// TIA Portal V18 export
FUNCTION "MotionController" : Void   // FC14, LAD
{ S7_Optimized_Access := 'TRUE' }
AUTHOR : HenriP
VERSION : 0.1
// stored: AutoNumber true, IsIECCheckEnabled false, SetENOAutomatically false, UDAEnableTagReadback false
   VAR_INPUT
      "E-STOP" : Bool;
      JogPBtn : Bool;
      JogNBtn : Bool;
      TargetRange : DInt;
      PosMax : DInt;
      PosMin : DInt;
      AxisColision : Bool;
      DoorSensor : Bool;
   END_VAR
   VAR_OUTPUT
      AxisOutput : Struct
         DriveEnabled : Bool;
         Ready : Bool;
         Warning : Bool;
         Fault : Bool;
         SupplyVoltPresent : Bool;
         ControlFCT_HMI : Bool;
         StateOPM : Int;
         HaltNotActive : Bool;
         AckStart : Bool;
         MC : Bool;
         AckTeach : Bool;
         DriveMoving : Bool;
         DragError : Bool;
         StandStillControl : Bool;
         HomingValid : Bool;
         ActualRecordNo : Int;
         RC1 : Bool;
         RCC : Bool;
         VelocityLimitReached : Bool;
         StrokeLimitReached : Bool;
         FunctionIsActive : Bool;
         ActualFunctionNumber : Int;
         ActualFunctionGroup : Int;
         ActualPosition : DInt;
         ActualVelocity : DInt;
         ActualForce : DInt;
         ActualRotRamp : DInt;
         ActualRotSpeed : DInt;
      END_STRUCT;
      TargetReached : Bool;
      Overange : Bool;
   END_VAR
   VAR_IN_OUT
      AxisInput : Struct
         EnableDrive : Bool;
         Stop : Bool;
         Halt : Bool;
         Brake : Bool;
         ResetFault : Bool;
         HMIAccessLocked : Bool;
         OPM : Int;
         StartTask : Bool;
         StartHoming : Bool;
         JogPos : Bool;
         JogNeg : Bool;
         TeachActValue : Bool;
         ClearRemPos : Bool;
         Relative : Bool;
         DeactivateStrokeLimit : Bool;
         ExecuteFunction : Bool;
         RecordNo : Int;
         SetFunctionNumber : Int;
         SetFunctionGroup : Int;
         SetValueVelocity : DInt;
         SetValuePosition : DInt;
         SetValueForceRamp : DInt;
         SetValueForce : DInt;
         SetValueRotRamp : DInt;
         SetValueRotSpeed : DInt;
      END_STRUCT;
      FestoDB : "FHPP_CTRL";
      TaskE : Bool;
      TaskM : Bool;
   END_VAR
   VAR_TEMP
      TargetDistance : DInt;
      ErrorValue : Int;
      Pos : DInt;
      PosAdd : DInt;
      PosSub : DInt;
      TaskEBis : Bool;
      JogPOv : DInt;
   END_VAR
   VAR_TEMP   // added for the SCL form of the ladder/FBD networks
      _w1 : Bool;
      _w2 : Bool;
   END_VAR
BEGIN

REGION Network 1: Enable Axis - Stop Control
   // For safety reason the Safety torque control is on a special loop , Emergency stop may move there too
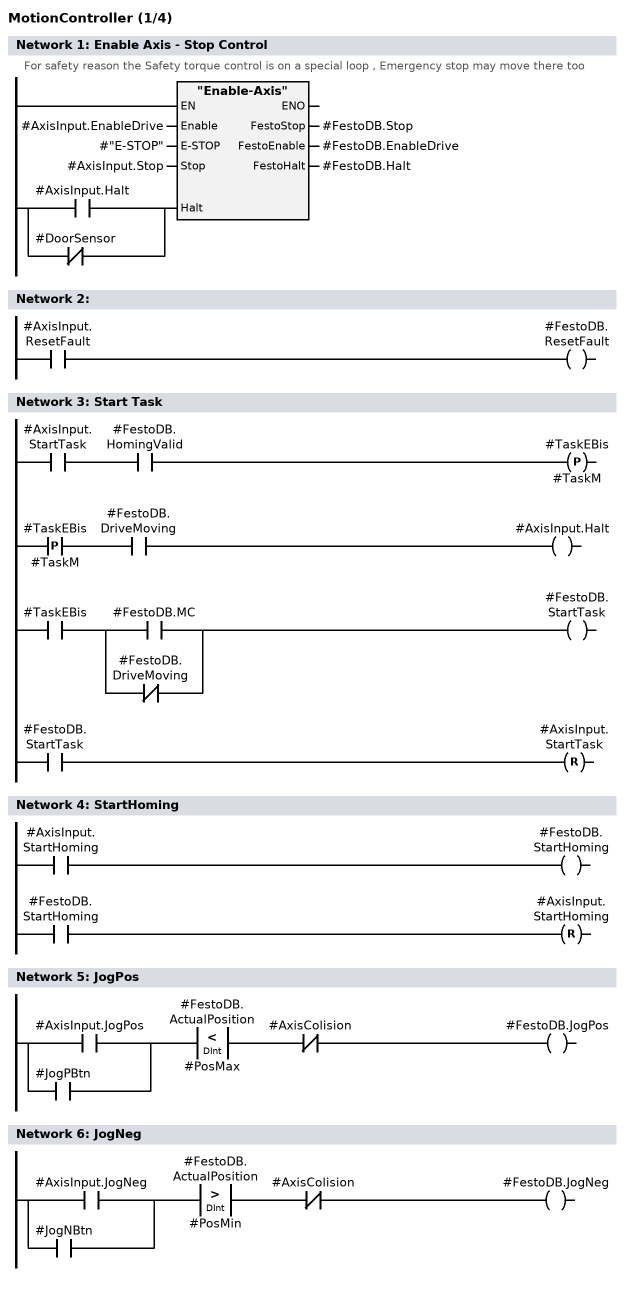
   RUNG wire#powerrail
      "Enable-Axis"(Halt := wire#w1, Enable := #AxisInput.EnableDrive, "E-STOP" := #"E-STOP", Stop := #AxisInput.Stop, FestoStop => #FestoDB.Stop, FestoEnable => #FestoDB.EnableDrive, FestoHalt => #FestoDB.Halt)
   END_RUNG
   RUNG wire#powerrail
      Contact( #AxisInput.Halt )
   END_RUNG wire#w1
   RUNG wire#powerrail
      I_Contact( #DoorSensor )
   END_RUNG wire#w1
   // the same network as SCL:
   "Enable-Axis"(Enable := #AxisInput.EnableDrive,
                 "E-STOP" := #"E-STOP",
                 Stop := #AxisInput.Stop,
                 Halt := #AxisInput.Halt OR NOT #DoorSensor,
                 FestoStop => #FestoDB.Stop,
                 FestoEnable => #FestoDB.EnableDrive,
                 FestoHalt => #FestoDB.Halt);
END_REGION

REGION Network 2
   RUNG wire#powerrail
      Contact( #AxisInput.ResetFault )
      Coil( #FestoDB.ResetFault )
   END_RUNG
   // the same network as SCL:
   #FestoDB.ResetFault := #AxisInput.ResetFault;
END_REGION

REGION Network 3: Start Task
   #_w1 := #AxisInput.StartTask AND #FestoDB.HomingValid;
   #TaskEBis := #_w1 AND NOT #TaskM;   // rising edge
   #TaskM := #_w1;
   #_w2 := #TaskEBis AND NOT #TaskM;   // rising edge of #TaskEBis
   #TaskM := #TaskEBis;
   #AxisInput.Halt := #_w2 AND #FestoDB.DriveMoving;
   #FestoDB.StartTask := #TaskEBis AND (#FestoDB.MC OR NOT #FestoDB.DriveMoving);
   IF #FestoDB.StartTask THEN #AxisInput.StartTask := FALSE; END_IF;
END_REGION

REGION Network 4: StartHoming
   RUNG wire#powerrail
      Contact( #AxisInput.StartHoming )
      Coil( #FestoDB.StartHoming )
   END_RUNG
   RUNG wire#powerrail
      Contact( #FestoDB.StartHoming )
      R_Coil( #AxisInput.StartHoming )
   END_RUNG
   // the same network as SCL:
   #FestoDB.StartHoming := #AxisInput.StartHoming;
   IF #FestoDB.StartHoming THEN #AxisInput.StartHoming := FALSE; END_IF;
END_REGION

REGION Network 5: JogPos
   RUNG wire#powerrail
      Contact( #AxisInput.JogPos )
      wire#w1
      { S7_Templates := "SrcType := DInt" } LT_Contact(in1 := #FestoDB.ActualPosition, in2 := #PosMax)
      I_Contact( #AxisColision )
      Coil( #FestoDB.JogPos )
   END_RUNG
   RUNG wire#powerrail
      Contact( #JogPBtn )
   END_RUNG wire#w1
   // the same network as SCL:
   #FestoDB.JogPos := (#AxisInput.JogPos OR #JogPBtn) AND (#FestoDB.ActualPosition < #PosMax) AND NOT #AxisColision;
END_REGION

REGION Network 6: JogNeg
   RUNG wire#powerrail
      Contact( #AxisInput.JogNeg )
      wire#w1
      { S7_Templates := "SrcType := DInt" } GT_Contact(in1 := #FestoDB.ActualPosition, in2 := #PosMin)
      I_Contact( #AxisColision )
      Coil( #FestoDB.JogNeg )
   END_RUNG
   RUNG wire#powerrail
      Contact( #JogNBtn )
   END_RUNG wire#w1
   // the same network as SCL:
   #FestoDB.JogNeg := (#AxisInput.JogNeg OR #JogNBtn) AND (#FestoDB.ActualPosition > #PosMin) AND NOT #AxisColision;
END_REGION

REGION Network 7: Relative Input Command
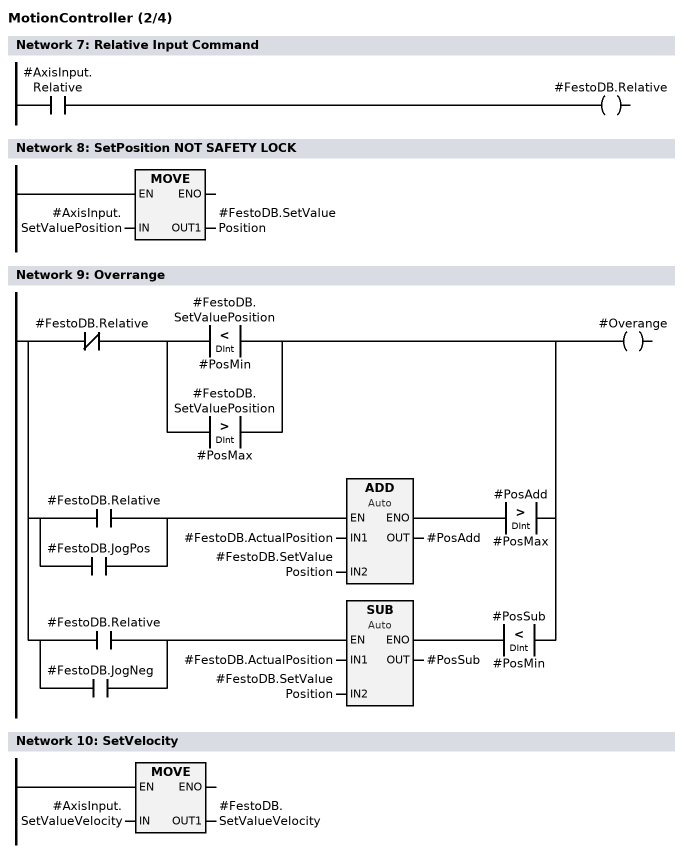
   RUNG wire#powerrail
      Contact( #AxisInput.Relative )
      Coil( #FestoDB.Relative )
   END_RUNG
   // the same network as SCL:
   #FestoDB.Relative := #AxisInput.Relative;
END_REGION

REGION Network 8: SetPosition NOT SAFETY LOCK
   RUNG wire#powerrail
      Move(in := #AxisInput.SetValuePosition, out1 => #FestoDB.SetValuePosition)
   END_RUNG
   // the same network as SCL:
   #FestoDB.SetValuePosition := #AxisInput.SetValuePosition;
END_REGION

REGION Network 9: Overrange
   RUNG wire#powerrail
      I_Contact( #FestoDB.Relative )
      wire#w1
      { S7_Templates := "SrcType := DInt" } LT_Contact(in1 := #FestoDB.SetValuePosition, in2 := #PosMin)
      wire#w2
      Coil( #Overange )
   END_RUNG
   RUNG wire#w1
      { S7_Templates := "SrcType := DInt" } GT_Contact(in1 := #FestoDB.SetValuePosition, in2 := #PosMax)
   END_RUNG wire#w2
   RUNG wire#powerrail
      Contact( #FestoDB.Relative )
      wire#w3
      Add(in1 := #FestoDB.ActualPosition, in2 := #FestoDB.SetValuePosition, out => #PosAdd)
      { S7_Templates := "SrcType := DInt" } GT_Contact(in1 := #PosAdd, in2 := #PosMax)
   END_RUNG wire#w2
   RUNG wire#powerrail
      Contact( #FestoDB.JogPos )
   END_RUNG wire#w3
   RUNG wire#powerrail
      Contact( #FestoDB.Relative )
      wire#w4
      Sub(in1 := #FestoDB.ActualPosition, in2 := #FestoDB.SetValuePosition, out => #PosSub)
      { S7_Templates := "SrcType := DInt" } LT_Contact(in1 := #PosSub, in2 := #PosMin)
   END_RUNG wire#w2
   RUNG wire#powerrail
      Contact( #FestoDB.JogNeg )
   END_RUNG wire#w4
   // the same network as SCL:
   #_w1 := #FestoDB.Relative OR #FestoDB.JogPos;
   IF #_w1 THEN #PosAdd := #FestoDB.ActualPosition + #FestoDB.SetValuePosition; END_IF;
   #_w2 := #FestoDB.Relative OR #FestoDB.JogNeg;
   IF #_w2 THEN #PosSub := #FestoDB.ActualPosition - #FestoDB.SetValuePosition; END_IF;
   #Overange := (NOT #FestoDB.Relative AND ((#FestoDB.SetValuePosition < #PosMin) OR (#FestoDB.SetValuePosition > #PosMax))) OR (#_w1 AND (#PosAdd > #PosMax)) OR (#_w2 AND (#PosSub < #PosMin));
END_REGION

REGION Network 10: SetVelocity
   RUNG wire#powerrail
      Move(in := #AxisInput.SetValueVelocity, out1 => #FestoDB.SetValueVelocity)
   END_RUNG
   // the same network as SCL:
   #FestoDB.SetValueVelocity := #AxisInput.SetValueVelocity;
END_REGION

REGION Network 11: Output Feedback
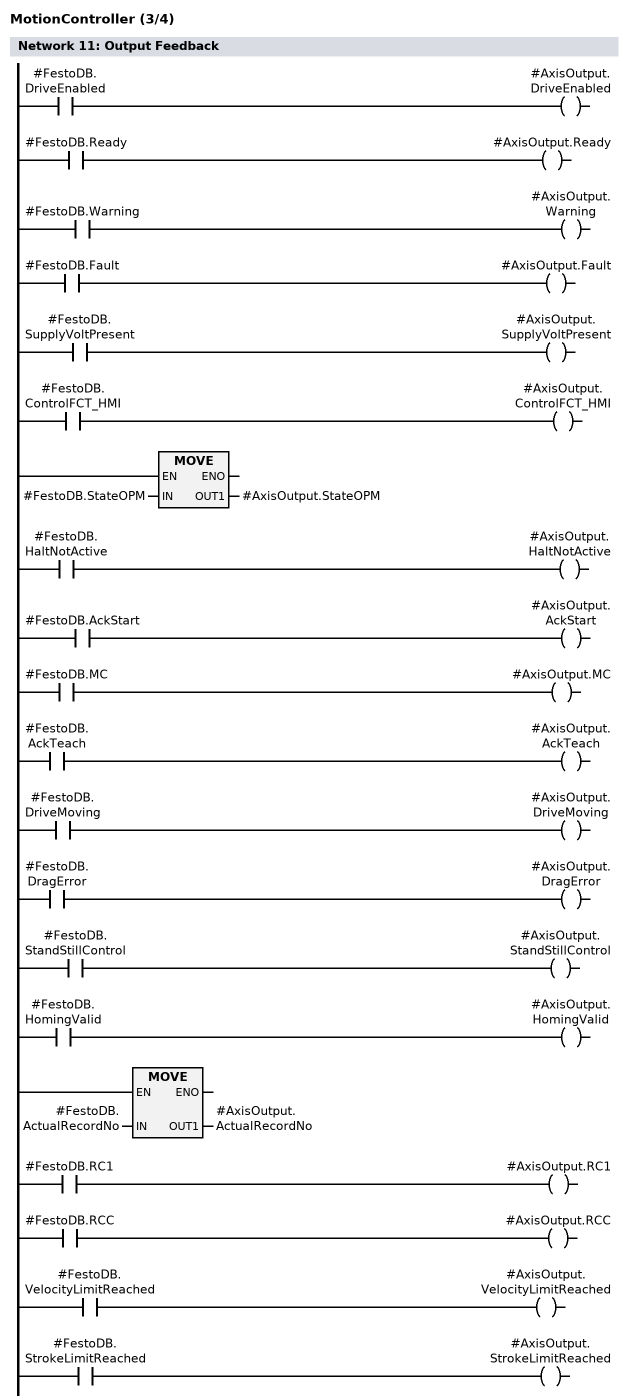
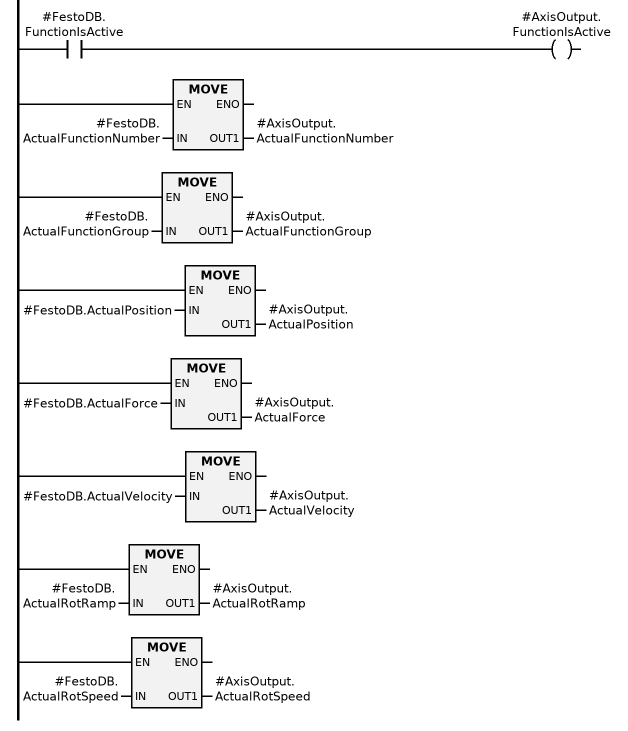
   RUNG wire#powerrail
      Contact( #FestoDB.DriveEnabled )
      Coil( #AxisOutput.DriveEnabled )
   END_RUNG
   RUNG wire#powerrail
      Contact( #FestoDB.Ready )
      Coil( #AxisOutput.Ready )
   END_RUNG
   RUNG wire#powerrail
      Contact( #FestoDB.Warning )
      Coil( #AxisOutput.Warning )
   END_RUNG
   RUNG wire#powerrail
      Contact( #FestoDB.Fault )
      Coil( #AxisOutput.Fault )
   END_RUNG
   RUNG wire#powerrail
      Contact( #FestoDB.SupplyVoltPresent )
      Coil( #AxisOutput.SupplyVoltPresent )
   END_RUNG
   RUNG wire#powerrail
      Contact( #FestoDB.ControlFCT_HMI )
      Coil( #AxisOutput.ControlFCT_HMI )
   END_RUNG
   RUNG wire#powerrail
      Move(in := #FestoDB.StateOPM, out1 => #AxisOutput.StateOPM)
   END_RUNG
   RUNG wire#powerrail
      Contact( #FestoDB.HaltNotActive )
      Coil( #AxisOutput.HaltNotActive )
   END_RUNG
   RUNG wire#powerrail
      Contact( #FestoDB.AckStart )
      Coil( #AxisOutput.AckStart )
   END_RUNG
   RUNG wire#powerrail
      Contact( #FestoDB.MC )
      Coil( #AxisOutput.MC )
   END_RUNG
   RUNG wire#powerrail
      Contact( #FestoDB.AckTeach )
      Coil( #AxisOutput.AckTeach )
   END_RUNG
   RUNG wire#powerrail
      Contact( #FestoDB.DriveMoving )
      Coil( #AxisOutput.DriveMoving )
   END_RUNG
   RUNG wire#powerrail
      Contact( #FestoDB.DragError )
      Coil( #AxisOutput.DragError )
   END_RUNG
   RUNG wire#powerrail
      Contact( #FestoDB.StandStillControl )
      Coil( #AxisOutput.StandStillControl )
   END_RUNG
   RUNG wire#powerrail
      Contact( #FestoDB.HomingValid )
      Coil( #AxisOutput.HomingValid )
   END_RUNG
   RUNG wire#powerrail
      Move(in := #FestoDB.ActualRecordNo, out1 => #AxisOutput.ActualRecordNo)
   END_RUNG
   RUNG wire#powerrail
      Contact( #FestoDB.RC1 )
      Coil( #AxisOutput.RC1 )
   END_RUNG
   RUNG wire#powerrail
      Contact( #FestoDB.RCC )
      Coil( #AxisOutput.RCC )
   END_RUNG
   RUNG wire#powerrail
      Contact( #FestoDB.VelocityLimitReached )
      Coil( #AxisOutput.VelocityLimitReached )
   END_RUNG
   RUNG wire#powerrail
      Contact( #FestoDB.StrokeLimitReached )
      Coil( #AxisOutput.StrokeLimitReached )
   END_RUNG
   RUNG wire#powerrail
      Contact( #FestoDB.FunctionIsActive )
      Coil( #AxisOutput.FunctionIsActive )
   END_RUNG
   RUNG wire#powerrail
      Move(in := #FestoDB.ActualFunctionNumber, out1 => #AxisOutput.ActualFunctionNumber)
   END_RUNG
   RUNG wire#powerrail
      Move(in := #FestoDB.ActualFunctionGroup, out1 => #AxisOutput.ActualFunctionGroup)
   END_RUNG
   RUNG wire#powerrail
      Move(in := #FestoDB.ActualPosition, out1 => #AxisOutput.ActualPosition)
   END_RUNG
   RUNG wire#powerrail
      Move(in := #FestoDB.ActualForce, out1 => #AxisOutput.ActualForce)
   END_RUNG
   RUNG wire#powerrail
      Move(in := #FestoDB.ActualVelocity, out1 => #AxisOutput.ActualVelocity)
   END_RUNG
   RUNG wire#powerrail
      Move(in := #FestoDB.ActualRotRamp, out1 => #AxisOutput.ActualRotRamp)
   END_RUNG
   RUNG wire#powerrail
      Move(in := #FestoDB.ActualRotSpeed, out1 => #AxisOutput.ActualRotSpeed)
   END_RUNG
   // the same network as SCL:
   #AxisOutput.DriveEnabled := #FestoDB.DriveEnabled;
   #AxisOutput.Ready := #FestoDB.Ready;
   #AxisOutput.Warning := #FestoDB.Warning;
   #AxisOutput.Fault := #FestoDB.Fault;
   #AxisOutput.SupplyVoltPresent := #FestoDB.SupplyVoltPresent;
   #AxisOutput.ControlFCT_HMI := #FestoDB.ControlFCT_HMI;
   #AxisOutput.StateOPM := #FestoDB.StateOPM;
   #AxisOutput.HaltNotActive := #FestoDB.HaltNotActive;
   #AxisOutput.AckStart := #FestoDB.AckStart;
   #AxisOutput.MC := #FestoDB.MC;
   #AxisOutput.AckTeach := #FestoDB.AckTeach;
   #AxisOutput.DriveMoving := #FestoDB.DriveMoving;
   #AxisOutput.DragError := #FestoDB.DragError;
   #AxisOutput.StandStillControl := #FestoDB.StandStillControl;
   #AxisOutput.HomingValid := #FestoDB.HomingValid;
   #AxisOutput.ActualRecordNo := #FestoDB.ActualRecordNo;
   #AxisOutput.RC1 := #FestoDB.RC1;
   #AxisOutput.RCC := #FestoDB.RCC;
   #AxisOutput.VelocityLimitReached := #FestoDB.VelocityLimitReached;
   #AxisOutput.StrokeLimitReached := #FestoDB.StrokeLimitReached;
   #AxisOutput.FunctionIsActive := #FestoDB.FunctionIsActive;
   #AxisOutput.ActualFunctionNumber := #FestoDB.ActualFunctionNumber;
   #AxisOutput.ActualFunctionGroup := #FestoDB.ActualFunctionGroup;
   #AxisOutput.ActualPosition := #FestoDB.ActualPosition;
   #AxisOutput.ActualForce := #FestoDB.ActualForce;
   #AxisOutput.ActualVelocity := #FestoDB.ActualVelocity;
   #AxisOutput.ActualRotRamp := #FestoDB.ActualRotRamp;
   #AxisOutput.ActualRotSpeed := #FestoDB.ActualRotSpeed;
END_REGION

REGION Network 12: TargetReached
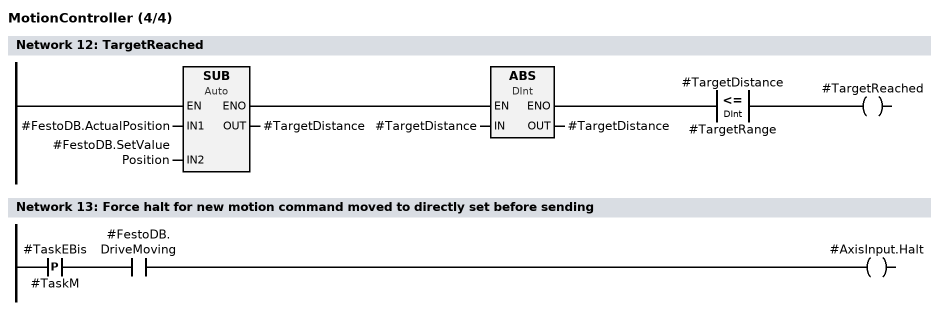
   RUNG wire#powerrail
      Sub(in1 := #FestoDB.ActualPosition, in2 := #FestoDB.SetValuePosition, out => #TargetDistance)
      { S7_Templates := "SrcType := DInt" } Abs(in := #TargetDistance, out => #TargetDistance)
      { S7_Templates := "SrcType := DInt" } LE_Contact(in1 := #TargetDistance, in2 := #TargetRange)
      Coil( #TargetReached )
   END_RUNG
   // the same network as SCL:
   #TargetDistance := #FestoDB.ActualPosition - #FestoDB.SetValuePosition;
   #TargetDistance := ABS(#TargetDistance);
   #TargetReached := #TargetDistance <= #TargetRange;
END_REGION

REGION Network 13: Force halt for new motion command moved to directly set before sending
   RUNG wire#powerrail
      P_Contact(operand := #TaskEBis, bit := #TaskM)
      Contact( #FestoDB.DriveMoving )
      Coil( #AxisInput.Halt )
   END_RUNG
   // the same network as SCL:
   #_w1 := #TaskEBis AND NOT #TaskM;   // rising edge of #TaskEBis
   #TaskM := #TaskEBis;
   #AxisInput.Halt := #_w1 AND #FestoDB.DriveMoving;
END_REGION
END_FUNCTION
